FUNCTION_BLOCK E_TRAIN (* Composite Function Block Type *)
  (* Standard: 61499-2 *)
  (* Version 0.0, 9/9/2026, macie, Schneider Electric, template *)
  PACKAGE Main;
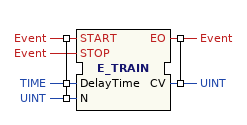
  EVENT_INPUT
    START WITH DelayTime, N; (* Initialization Request *)
    STOP; (* Normal Execution Request *)
  END_EVENT
  EVENT_OUTPUT
    EO WITH CV; (* Execution Confirmation *)
  END_EVENT
  VAR_INPUT
    DelayTime : TIME := T#0s;
    N : UINT := 0;
  END_VAR
  VAR_OUTPUT
    CV : UINT := 0; (* Output event qualifier *)
  END_VAR
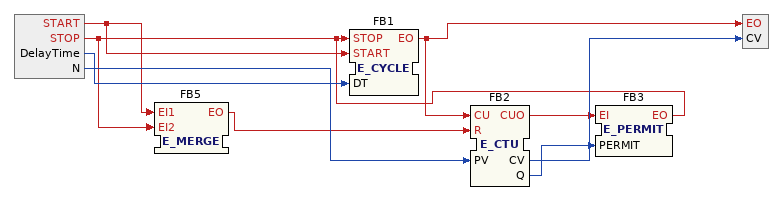
  FBS
    FB1 : E_CYCLE;
    FB2 : E_CTU;
    FB3 : E_PERMIT;
    FB5 : E_MERGE;
  END_FBS
  EVENT_CONNECTIONS
    STOP TO FB1.STOP;
    START TO FB1.START;
    FB1.EO TO EO;
    FB1.EO TO FB2.CU;
    FB2.CUO TO FB3.EI;
    FB3.EO TO FB1.STOP;
    START TO FB5.EI1;
    STOP TO FB5.EI2;
    FB5.EO TO FB2.R;
  END_CONNECTIONS
  DATA_CONNECTIONS
    DelayTime TO FB1.DT;
    FB2.CV TO CV;
    N TO FB2.PV;
    FB2.Q TO FB3.PERMIT;
  END_CONNECTIONS
END_FUNCTION_BLOCK
